(* IEC 61131-3 sources: ElnaAutomator/ExampleProject/Programs, 1 file *)

(* ---- program0.st ---- *)
PROGRAM program0

VAR
	Var0 : DINT;
END_VAR

Var0 := 1;
